(* CODESYS project PLC_Project_Codesys.export

Project tree, tasks and I/O mapping:
  Device : CODESYS Control Win V3, 3S - Smart Software Solutions GmbH, version 3.5.14.20
    application Application
      libraries: Standard, * (System)
      task MainTask (cyclic, interval t#20ms, priority 1) calls PLC_PRG
      program PLC_PRG [LD]
    Ethernet : Ethernet, 3S - Smart Software Solutions GmbH, version 3.5.14.0
        settings: IPAddress = [192,168,15,80]; SubnetMask = [255,255,255,0]; GatewayAddress = [192,168,15,1]; MACAddress = [16#E8,16#FB,16#1C,16#A0,16#69,16#3F]; NetworkInterfaceName = 'Wi-Fi'; NetworkInterfaceName = "Wi-Fi"; SaveCommunicationSettings = FALSE
      ModbusTCP_Slave_Device : ModbusTCP Slave Device, 3S - Smart Software Solutions GmbH, version 3.5.14.0
          settings: Unit-ID = 1; StartAdresses.Coils = 1
          input  Application.PLC_PRG.I_VN : BOOL  // Inputs.Inputs.Bit0
          input  Application.PLC_PRG.RELAY : BOOL  // Inputs.Inputs.Bit1
          input  Application.PLC_PRG.TU_ON : BOOL  // Inputs.Inputs.Bit2
          input  Application.PLC_PRG.TU_OFF : BOOL  // Inputs.Inputs.Bit3
          input  Application.PLC_PRG.TU : BOOL  // Inputs.Inputs.Bit4
          input  Application.PLC_PRG.TU_TRIP : BOOL  // Inputs.Inputs.Bit5
          input  Application.PLC_PRG.TempChiller : BOOL  // Inputs.Inputs.Bit6
          input  Application.PLC_PRG.P_PUMP : BOOL  // Inputs.Inputs.Bit7
          input  Application.PLC_PRG.DISC_PRESS : BOOL  // Inputs.Inputs.Bit8
          input  Application.PLC_PRG.TEMP_COMP : BOOL  // Inputs.Inputs.Bit9
          input  Application.PLC_PRG.TU_TRIP_S : BOOL  // Inputs.Inputs.Bit10
          input  Application.PLC_PRG.LOGIC_1 : BOOL  // Inputs.Inputs.Bit11
          input  Application.PLC_PRG.LOGIC_2 : BOOL  // Inputs.Inputs.Bit12
          input  Application.PLC_PRG.LOGIC_3 : BOOL  // Inputs.Inputs.Bit13
          input  Application.PLC_PRG.LOGIC_4 : BOOL  // Inputs.Inputs.Bit14
          input  Application.PLC_PRG.TON_0.Q : BOOL  // Inputs.Inputs.Bit15
          input  Application.PLC_PRG.DJ1 : BOOL  // Inputs.Inputs.Bit0
          input  Application.PLC_PRG.DJ1_OFF : BOOL  // Inputs.Inputs.Bit1
          input  Application.PLC_PRG.DJ1_ON : BOOL  // Inputs.Inputs.Bit2
          input  Application.PLC_PRG.DJ2 : BOOL  // Inputs.Inputs.Bit3
          input  Application.PLC_PRG.DJ2_OFF : BOOL  // Inputs.Inputs.Bit4
          input  Application.PLC_PRG.DJ2_ON : BOOL  // Inputs.Inputs.Bit5
          input  Application.PLC_PRG.DJ3 : BOOL  // Inputs.Inputs.Bit6
          input  Application.PLC_PRG.DJ3_OFF : BOOL  // Inputs.Inputs.Bit7
          input  Application.PLC_PRG.DJ3_ON : BOOL  // Inputs.Inputs.Bit8
          input  Application.PLC_PRG.CHILLER : BOOL  // Inputs.Inputs.Bit9
          input  Application.PLC_PRG.PUMP : BOOL  // Inputs.Inputs.Bit10
          input  Application.PLC_PRG.COMPRESSOR : BOOL  // Inputs.Inputs.Bit11
          input  Application.PLC_PRG.PLC : BOOL  // Inputs.Inputs.Bit12
          unmapped channels: Inputs, Outputs
*)

// Device/Application/PLC_PRG
PROGRAM PLC_PRG
VAR
	//Trip Unit Logic
	I_VN: BOOL; 		//It signal come from trip unit readings
	TON_0: TON;			//Timer counter to logic 1
	LOGIC_1: BOOL;		//Output logic 1
	//Relay's signal
	RELAY: BOOL;		//It Signal from Relay's digital output
	//Trip Unit States
	TU_ON: BOOL;
	TU_OFF: BOOL;
	TU: BOOL;
	TU_TRIP_S: BOOL; 	//input to trip
	TU_TRIP: BOOL;		//output to trip	
	//CAG Logicals
	TempChiller: BOOL;	//Temperature from chiller - Logical from Supervisory
	LOGIC_2: BOOL;		// Output logic 2
	P_PUMP: BOOL;		// Chiller's Pump Pressure - Logical from Supervisory
	LOGIC_3: BOOL;		// Output Logic 3
	//Compressor Logicals
	DISC_PRESS: BOOL;	// Compressor discharge pressure - Logical from Supervisory
	TEMP_COMP: BOOL;	// Compressor Teperature - Logical from Supervisory
	LOGIC_4: BOOL;		// Output Logic 4
	//Breakers
	DJ1_ON: BOOL;		//DJ1 CAG (Chiller and Pump) Breaker
	DJ1_OFF: BOOL;
	DJ1: BOOL;
	DJ2_ON: BOOL;		//Compressor breaker
	DJ2_OFF: BOOL;
	DJ2: BOOL;
	DJ3_ON: BOOL;		//CLP Breaker
	DJ3_OFF: BOOL;
	DJ3: BOOL;
	//System Equipments (devices)
	CHILLER: BOOL;
	PUMP: BOOL;
	COMPRESSOR: BOOL;
	PLC: BOOL;
	new: BOOL;
	TU_OFF2: BOOL;
END_VAR
VAR // added by the converter: edge detectors and wires of the graphical bodies
    _w1, _w2, _w3 : BOOL;
END_VAR

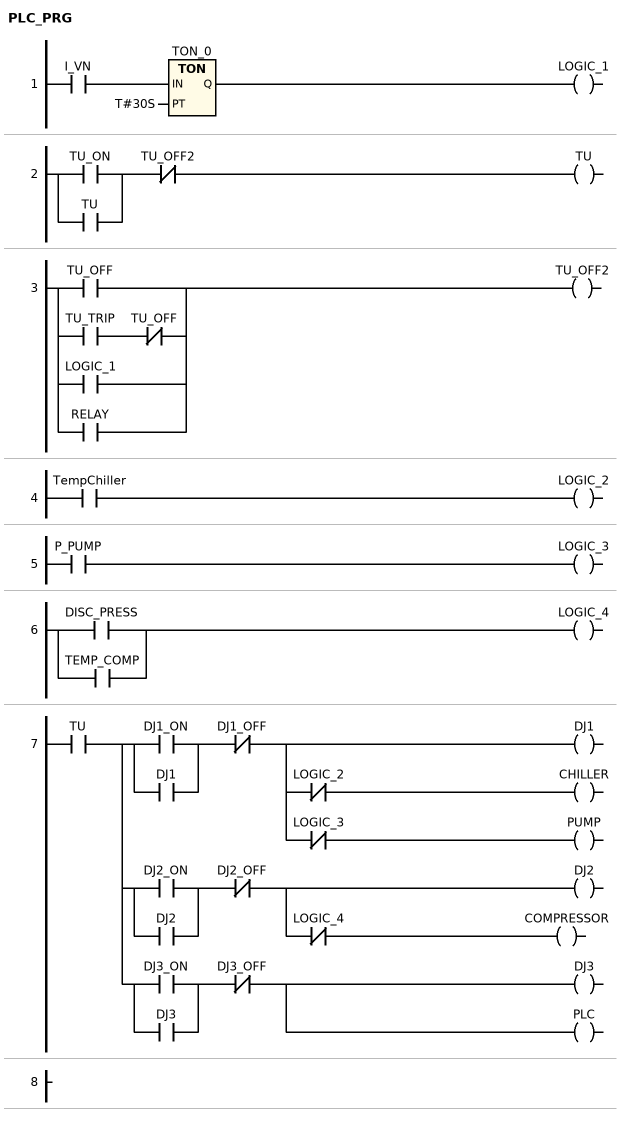
// NETWORK 1
TON_0(IN := I_VN, PT := T#30S); // TON
LOGIC_1 := TON_0.Q;

// NETWORK 2
TU := (TU_ON OR TU) AND NOT TU_OFF2;

// NETWORK 3
TU_OFF2 := TU_OFF OR TU_TRIP AND NOT TU_OFF OR LOGIC_1 OR RELAY;

// NETWORK 4
LOGIC_2 := TempChiller;

// NETWORK 5
LOGIC_3 := P_PUMP;

// NETWORK 6
LOGIC_4 := DISC_PRESS OR TEMP_COMP;

// NETWORK 7
_w1 := TU AND (DJ1_ON OR DJ1) AND NOT DJ1_OFF;
DJ1 := _w1;
CHILLER := _w1 AND NOT LOGIC_2;
PUMP := _w1 AND NOT LOGIC_3;
_w2 := TU AND (DJ2_ON OR DJ2) AND NOT DJ2_OFF;
DJ2 := _w2;
COMPRESSOR := _w2 AND NOT LOGIC_4;
_w3 := TU AND (DJ3_ON OR DJ3) AND NOT DJ3_OFF;
DJ3 := _w3;
PLC := _w3;

// NETWORK 8

END_PROGRAM
